INTERFACE I_Diverter

PROPERTY bError : BOOL
GET
END_GET
END_PROPERTY

PROPERTY bLiftUp : BOOL
GET
END_GET
END_PROPERTY

PROPERTY bTravelMotorRun : BOOL
GET
END_GET
END_PROPERTY

PROPERTY eState : E_DiverterState
GET
END_GET
END_PROPERTY

METHOD M_Divert
VAR_INPUT
END_VAR
END_METHOD

METHOD M_Stop
VAR_INPUT
END_VAR
END_METHOD

END_INTERFACE

(* stored: Version 1.1.0.1, ProductVersion 3.1.4024.16
   Itf I_Diverter: Id {84cfe86d-85ae-4d1c-a69c-ff269d5b2ee5}
   Property bError: Id {3e4f5a6b-c7d8-9012-4567-123456789012}
   Get Get: Id {4f5a6b7c-d8e9-0123-5678-234567890123}
   Property bLiftUp: Id {5a6b7c8d-e9f0-1234-6789-345678901234}
   Get Get: Id {6b7c8d9e-f0a1-2345-7890-456789012345}
   Property bTravelMotorRun: Id {7c8d9e0f-a1b2-3456-8901-567890123456}
   Get Get: Id {8d9e0f1a-b2c3-4567-9012-678901234567}
   Property eState: Id {9e0f1a2b-c3d4-5678-0123-789012345678}
   Get Get: Id {0f1a2b3c-d4e5-6789-1234-890123456789}
   Method M_Divert: Id {1a2b3c4d-e5f6-7890-2345-901234567890}
   Method M_Stop: Id {2b3c4d5e-f6a7-8901-3456-012345678901} *)
